TEXTLIST TelemetryConfigTextList
  0 = 'Temperatures: M1'
  1 = 'Temperatures: Mirror cell'
  2 = 'Temperatures: M2'
  3 = 'Temperatures: M2 electronics'
  4 = 'Temperatures: Top tube'
  5 = 'Temperatures: Centre tube'
  6 = 'Temperatures: Fork'
  7 = 'Temperatures: Nasmyth air'
  8 = 'Temperatures: REM cabinet'
  9 = 'Temperatures: RPM cabinet'
  10 = 'Temperatures: HERMES telescope adapter'
  11 = 'Temperatures: Top air'
  12 = 'Temperatures: Inside tube'
  13 = 'Relative humidities: Top air'
  14 = 'Relative humidities: Inside tube'
  15 = 'Dewpoints: Top air'
  16 = 'Dewpoints: Inside tube'
  17 = 'Accelerometers: Tube X angle'
  18 = 'Accelerometers: Tube Y angle'
   = ''
END_TEXTLIST

(* stored: Version 1.1.0.1, ProductVersion 3.1.4018.5
   TextList TelemetryConfigTextList: Id {c6ea840f-b8be-4c79-a673-a849bf3d16c4} *)
